{attribute 'linkalways'} 
{attribute 'no_explicit_call' := 'This FB is a CLASS and must be accessed using methods or properties'}
{attribute 'enable_dynamic_creation'}
FUNCTION_BLOCK _ETcVnClusteringAlgorithm EXTENDS EnumDatatypeBase
VAR
	localData : ETcVnClusteringAlgorithm;
	activeData : REFERENCE TO ETcVnClusteringAlgorithm;
	enumBaseDatatype : _DINT(localData);
END_VAR

METHOD PRIVATE AddLocalEnumeration
VAR_INPUT
	Enumeration : T_MAXSTRING;
	Value : ETcVnClusteringAlgorithm;
END_VAR
AddEnumeration(Enumeration, Value);
END_METHOD

PROPERTY PUBLIC Address : PVOID
GET
Address := ADR(activeData);
END_GET
END_PROPERTY

METHOD PUBLIC ClearReference
VAR_INPUT
END_VAR
activeData REF= localData;
SetBaseDatatypeReference();
END_METHOD

METHOD PUBLIC Clone : I_Datatype
VAR
    pClone : POINTER TO _ETcVnClusteringAlgorithm;
END_VAR
pClone := __NEW(_ETcVnClusteringAlgorithm(InitialValue := Value));
Clone := pClone^;
END_METHOD

METHOD FB_init : BOOL
VAR_INPUT
	bInitRetains : BOOL; // if TRUE, the retain variables are initialized (warm start / cold start)
	bInCopyCode : BOOL;  // if TRUE, the instance afterwards gets moved into the copy code (online change)
	InitialValue : ETcVnClusteringAlgorithm;
END_VAR
localData := InitialValue;
AddBaseDatatype(enumBaseDatatype);
ClearReference();

AddLocalEnumeration('TCVN_CA_KMEANSPP', ETcVnClusteringAlgorithm.TCVN_CA_KMEANSPP);
AddLocalEnumeration('TCVN_CA_LBG', ETcVnClusteringAlgorithm.TCVN_CA_LBG);
END_METHOD

PROPERTY PUBLIC Identifier : T_MAXSTRING
GET
Identifier := 'ETcVnClusteringAlgorithm';
END_GET
END_PROPERTY

METHOD IsEnumeratorValueEqual : BOOL
VAR_INPUT
	Enumerator : I_KeyValueForwardEnumerator;
END_VAR
VAR
	storedValue : ETcVnClusteringAlgorithm;
END_VAR
IF NOT Enumerator.TryGet(storedValue) THEN
	RETURN;
END_IF

IsEnumeratorValueEqual := storedValue = activeData;
END_METHOD

METHOD PUBLIC MakeReferenceTo
VAR_INPUT
	ReferenceTarget : REFERENCE TO ETcVnCalibrationPatternOrigin;
END_VAR
activeData REF= ReferenceTarget;
SetBaseDatatypeReference();
END_METHOD

METHOD PROTECTED SetBaseDatatypeReference
VAR_INPUT
END_VAR
enumBaseDatatype.MakeReferenceTo(activeData);
END_METHOD

PROPERTY PUBLIC Size : UDINT
GET
Size := SIZEOF(activeData);
END_GET
END_PROPERTY

METHOD TryMakeReferenceTo : BOOL
VAR_INPUT
	Target : I_Datatype;
END_VAR
VAR
	pTargetData : POINTER TO ETcVnClusteringAlgorithm;
END_VAR
IF NOT IsEquivalentTo(Target) THEN
	RETURN;
END_IF

pTargetData := Target.Address;
activeData REF= pTargetData^;
SetBaseDatatypeReference();
TryMakeReferenceTo := TRUE;
END_METHOD

PROPERTY PUBLIC Value : ETcVnClusteringAlgorithm
GET
Value := activeData;
END_GET
SET
activeData := Value;
END_SET
END_PROPERTY

END_FUNCTION_BLOCK

(* stored: Version 1.1.0.1, ProductVersion 3.1.4024.13
   POU _ETcVnClusteringAlgorithm: Id {276c8f38-e538-44c5-92df-6832fa0ee740}, SpecialFunc None
   Folder Core: Id {774c985c-b289-071c-00a4-58ca3fa1ff1c}
   Folder Protected: Id {9aee7715-bb06-0789-130c-2e9029ce20ad}
   Folder Customize: Id {54db5caf-90b3-09b1-356f-325f0e8d9a11}
   Folder Constructor: Id {2750bd5b-925e-4f50-9bbd-f47f1b52f223}
   Folder Private: Id {343b4180-5443-4fdf-82e4-5ea54836fa1e}
   Folder Protected: Id {af4b0071-04d4-4562-b7d7-a62fe10f127b}
   Method AddLocalEnumeration: Id {dcb45ecd-8097-4fc7-9a1c-e113ebb66a58}
   Property Address: Id {cd1fe1de-4646-0e97-1f63-2ea093e5db36}
   Get Get: Id {b21f5a59-9fb2-0b3f-078b-42a84a5edf4b}
   Method ClearReference: Id {63a953b9-6bf4-0503-2865-0db492d9e5db}
   Method Clone: Id {651dcbd4-1229-43e7-a64b-aacca98bc188}
   Method FB_init: Id {93105a62-b495-409d-b5a7-185cb3c463c9}
   Property Identifier: Id {fd71f75c-89f6-48f9-b415-7fd4863854e7}
   Get Get: Id {1b57410b-5ba0-4cf1-8101-cbfb638fbc5f}
   Method IsEnumeratorValueEqual: Id {1e4ce020-7464-446a-a323-8e2a8702e02c}
   Method MakeReferenceTo: Id {40d6fd12-6339-4332-a859-e95dcd6c11e8}
   Method SetBaseDatatypeReference: Id {a5744a20-13ad-02de-12e7-278eed9ff415}
   Property Size: Id {a62aa8ca-66f1-07c9-33b9-5e53d2d192ba}
   Get Get: Id {5f7e356e-cdfb-0bab-2e44-c5a55002d859}
   Method TryMakeReferenceTo: Id {ca39e4f5-131b-40a4-89ff-98d4aba524a1}
   Property Value: Id {364101c0-b561-42ec-817e-ef4735290591}
   Get Get: Id {8b3055b2-921b-4462-baec-5116c031defa}
   Set Set: Id {e7693a63-d9e7-41ff-add3-ec707427c854} *)
